TYPE STATE:
    STRUCT
        curTime: LREAL;
        dvar_M_g2_aut_z AT %Q*: DINT;
    END_STRUCT
END_TYPE

(* stored: ProductVersion 3.1.0.18, Version 1.1.0.1 *)
